// TIA Portal V20 export
TYPE "LER_typeRadiusMeasureConfiguration"
// stored: Access Published
   STRUCT
      Offset : LReal;
      DecimalPoint : Int;
   END_STRUCT;
END_TYPE
